FUNCTION_BLOCK BoolValuesTest EXTENDS TcUnit.FB_TestSuite

FalseBoolValue();
TrueBoolValue();

METHOD FalseBoolValue : BOOL
VAR
	value : FalseBoolValue;
END_VAR
TcUnit.TEST('Get false bool value');

AssertEquals_BOOL(
	Expected := FALSE,
	Actual := value.Value,
	Message := 'FalseBoolValue should return FALSE value');

TEST_FINISHED();
END_METHOD

METHOD TrueBoolValue : BOOL
VAR
	value : TrueBoolValue;
END_VAR
TcUnit.TEST('Get true bool value');

AssertEquals_BOOL(
	Expected := TRUE,
	Actual := value.Value,
	Message := 'TrueBoolValue should return TRUE value');

TEST_FINISHED();
END_METHOD

END_FUNCTION_BLOCK

(* stored: Version 1.1.0.1, ProductVersion 3.1.4024.12
   POU BoolValuesTest: Id {191f85c8-662c-078c-39b8-d20047e840af}, SpecialFunc None
   Method FalseBoolValue: Id {955706dd-0957-06a9-0489-b8163ccdabe0}
   Method TrueBoolValue: Id {1d34fa66-d939-0afb-028e-f5eba1317d2c} *)
